// TIA Portal project "MABFactoryIO_Project" (V18)
// TIA Portal - Factory IO

(* hardware
DEVICE "S71500/ET200MP-Station_1"  S7-1500 station
   slot 0: "Profilschiene_0"  Rack  6ES7 590-1***0-0AA0
   slot 1: "PLC_1"  CPU 1517-3 PN/DP  6ES7 517-3AP00-0AB0  V2.6
      slot 3: "CPU-Display_1"  6ES7591-1BA00-0AA0
      slot 32768: "PROFINET-Schnittstelle_1"  X1
         slot 32769: "Port_1"  X1 P1
         slot 32770: "Port_2"  X1 P2
      slot 33024: "PROFINET interface_1"  X2
      slot 33280: "DP interface_1"  X3
   slot 2: "AI 8xU/I/RTD/TC ST_1"  AI 8xU/I/RTD/TC ST  6ES7 531-7KF00-0AB0  V2.0
   slot 3: "AI 8xU/I/RTD/TC ST_2"  AI 8xU/I/RTD/TC ST  6ES7 531-7KF00-0AB0  V2.0
   slot 4: "AI 8xU/I/RTD/TC ST_3"  AI 8xU/I/RTD/TC ST  6ES7 531-7KF00-0AB0  V2.0
   slot 5: "AI 8xU/I/RTD/TC ST_4"  AI 8xU/I/RTD/TC ST  6ES7 531-7KF00-0AB0  V2.0
   slot 6: "DI 16x24VDC BA_1"  DI 16x24VDC BA  6ES7 521-1BH10-0AA0  V1.0
*)

// ===== PLC "PLC_1"  CPU 1517-3 PN/DP =====

VAR_GLOBAL   // PLC tag table "Standard-Variablentabelle"
   "BC-L0" AT %Q10.0 : Bool;
   "BC-L1.1" AT %Q10.1 : Bool;
   "BC-L2" AT %Q10.3 : Bool;
   "BC-L3" AT %Q10.4 : Bool;
   "BC-L4" AT %Q10.5 : Bool;
   "BCS-L0" AT %Q10.6 : Bool;
   "BCS-L1" AT %Q10.7 : Bool;
   "BCC-L0" AT %Q11.0 : Bool;
   "BC-R0" AT %Q11.1 : Bool;
   "BC-R1.1" AT %Q11.2 : Bool;
   "BC-R2" AT %Q11.4 : Bool;
   "BC-R3" AT %Q11.5 : Bool;
   "BCS-R0" AT %Q11.6 : Bool;
   "BCS-R1" AT %Q11.7 : Bool;
   "BCC-R0" AT %Q12.0 : Bool;
   "Conveyor_SR" AT %M10.0 : Bool;
   "Start_Button" AT %I0.0 : Bool;
   "Stop_Button" AT %I0.1 : Bool;
   "BluePileUp" AT %I5.0 : Bool;
   "GreenPileUp" AT %I5.1 : Bool;
   "GreenRawSensor" AT %I4.7 : Bool;
   "BluePileReset" AT %I4.6 : Bool;
   "BC-L1.2" AT %Q10.2 : Bool;
   "BC-R1.2" AT %Q11.3 : Bool;
   "PusherLımıt" AT %I5.2 : Bool;
   "GreenSequenceSensor" AT %I5.3 : Bool;
   "BlueLineSR" AT %M10.1 : Bool;
   "BlueSetter" AT %M1.0 : Bool;
   "GreenLineSR" AT %M10.2 : Bool;
   "GreenSetter" AT %M1.1 : Bool;
   "PusherRight" AT %Q5.0 : Bool;
   "GreenSubline" AT %Q5.1 : Bool;
   "RightLaneBlock" AT %M3.0 : Bool;
   "IsBusy" AT %M3.1 : Bool;
   "SortSR" AT %M10.3 : Bool;
   "SortSR_" AT %M10.4 : Bool;
   "BACUncontrolled" AT %Q3.0 : Bool;
   "BACSBL" AT %Q3.2 : Bool;
   "BSBLeft" AT %Q3.5 : Bool;
   "BACLoadBeltLeft" AT %Q3.3 : Bool;
   "BACLoadBeltRight" AT %Q3.4 : Bool;
   "BACSBR" AT %Q3.1 : Bool;
   "BlueSubline" AT %Q5.2 : Bool;
   "MachineCenterSR" AT %M10.5 : Bool;
   "Machine0" AT %Q0.0 : Bool;
   "Machine1" AT %Q0.1 : Bool;
   "Machine2" AT %Q0.2 : Bool;
   "Machine3" AT %Q0.3 : Bool;
   "Machine0ProduceLids" AT %Q0.4 : Bool;
   "Machine1ProduceLids" AT %Q0.5 : Bool;
   "GreenPileReset" AT %I4.5 : Bool;
   "GreenClosePrevent" AT %I4.4 : Bool;
   "BlueClosePrevent" AT %I4.3 : Bool;
   "MCIsBusy_0" AT %I1.0 : Bool;
   "MCIsBusy_1" AT %I1.1 : Bool;
   "MCIsBusy_2" AT %I1.2 : Bool;
   "MCIsBusy_3" AT %I1.3 : Bool;
   "LPLid_SR" AT %M10.6 : Bool;
   "LPBase_SR" AT %M10.7 : Bool;
   "DiffClampLid" AT %I1.4 : Bool;
   "DiffClampBase" AT %I1.5 : Bool;
   "LPBaseClamped" AT %I1.6 : Bool;
   "LPLidClamped" AT %I1.7 : Bool;
   "LPBaseClamp" AT %Q0.6 : Bool;
   "LPLidClamp" AT %Q0.7 : Bool;
   "TwoAxisDETECT" AT %I2.0 : Bool;
   "TwoAxisDOWN" AT %Q1.0 : Bool;
   "TwoAxisGRAB" AT %Q1.1 : Bool;
   "TwoAxisSR" AT %M11.0 : Bool;
   "LeftPositionerInLim" AT %I2.1 : Bool;
   "TwoAxisFRWD" AT %Q1.2 : Bool;
   "TwoAxisX" AT %I2.2 : Bool;
   "TwoAxisZ" AT %I2.3 : Bool;
   "TwoAxisUPDOWN" AT %I11.1 : Bool;
   "XlimReached" AT %M3.2 : Bool;
   "TwoAxisConnection" AT %M11.2 : Bool;
   "ConnectionComplete" AT %M3.3 : Bool;
   "TwoAxGrabbed" AT %M3.4 : Bool;
   "TwoAxisXSR" AT %M11.1 : Bool;
   "CapTwoAxinPos" AT %I2.4 : Bool;
   "LPRaise" AT %Q1.3 : Bool;
   "LastSR" AT %M11.4 : Bool;
   "CapFullPasse" AT %I2.5 : Bool;
   "AssemblerConvSR" AT %M11.5 : Bool;
   "ACUncontrolled" AT %Q2.0 : Bool;
   "ACFeedBelt" AT %Q2.1 : Bool;
   "ACSBL" AT %Q2.2 : Bool;
   "ACSBR" AT %Q2.3 : Bool;
   "SB_SR" AT %M11.6 : Bool;
   "ACLoadBeltLeft" AT %Q2.4 : Bool;
   "ACLoadBeltRight" AT %Q2.5 : Bool;
   "SBLeft" AT %Q2.6 : Bool;
   "SBRight" AT %Q2.7 : Bool;
   "DiffSBLeft" AT %I2.6 : Bool;
   "DiffSBRight" AT %I2.7 : Bool;
   "CapLoadPassed" AT %I3.0 : Bool;
   "ResetDelay" AT %M11.3 : Bool;
   "LaneFilled" AT %M3.5 : Bool;
   "AssemblerLoaded" AT %M3.6 : Bool;
   "CapBasePassed" AT %I3.1 : Bool;
   "BlueLidSR" AT %M12.0 : Bool;
   "BlueBaseSR" AT %M12.1 : Bool;
   "BlueGrabSR" AT %M12.2 : Bool;
   "BTwoAxForw" AT %M12.3 : Bool;
   "BDiffClampLid" AT %I6.0 : Bool;
   "BDiffClampBase" AT %I6.1 : Bool;
   "BRPBaseClamp" AT %I6.3 : Bool;
   "BLPLidClamped" AT %I6.2 : Bool;
   "BTwoAxDETECT" AT %I6.4 : Bool;
   "BTwoAxisX" AT %I6.5 : Bool;
   "BTwoAxisZ" AT %I6.6 : Bool;
   "BCapFullPassed" AT %I6.7 : Bool;
   "BTwoAxGRAB" AT %Q6.0 : Bool;
   "BRPClamp" AT %Q6.2 : Bool;
   "BLPLidClamp" AT %Q6.1 : Bool;
   "BTwoAxDOWN" AT %Q6.3 : Bool;
   "BTwoAxisFRWD" AT %Q6.4 : Bool;
   "BRPRise" AT %Q6.5 : Bool;
   "BSConvSR" AT %M13.0 : Bool;
   "BAConv_Filled" AT %M13.1 : Bool;
   "BAssemblerLoaded" AT %M3.7 : Bool;
   "BCapLidPassed" AT %I7.1 : Bool;
   "BCapBasePassed" AT %I7.0 : Bool;
   "BSBRight" AT %Q3.6 : Bool;
   "BDiffSBLeft" AT %I7.2 : Bool;
   "BDiffSBRight" AT %I7.3 : Bool;
   "R0 Reset" AT %I0.2 : Bool;
   "Tag_1" AT %M12.7 : Bool;
   "PalletizerSR" AT %M12.4 : Bool;
   "PalletizerPushSR" AT %M12.5 : Bool;
   "DiffPalletizerEntry" AT %I8.0 : Bool;
   "CapPalletizerİnLine" AT %I8.1 : Bool;
   "PalletizerPushLimit" AT %I8.2 : Bool;
   "PalletizerBelt+" AT %Q8.0 : Bool;
   "PalletizerPush" AT %Q8.1 : Bool;
   "CapPalletizerPushİnimit" AT %I8.3 : Bool;
   "CapProdSR" AT %M12.6 : Bool;
   "PalletizerClamped" AT %I8.4 : Bool;
   "PalletizerClamp" AT %Q8.2 : Bool;
END_VAR

// folder: Assembling Operations/BlueProductAssemblyLine

DATA_BLOCK "BlueAssemblerConveyor_DB"   // DB15
{ S7_Optimized_Access := 'TRUE' }
VERSION : 0.1
// stored: InstanceOfName BlueAssemblerConveyor
"BlueAssemblerConveyor"
BEGIN
END_DATA_BLOCK

DATA_BLOCK "BlueAssembler_DB"   // DB16
{ S7_Optimized_Access := 'TRUE' }
VERSION : 0.1
// stored: InstanceOfName BlueAssembler
"BlueAssembler"
BEGIN
END_DATA_BLOCK

DATA_BLOCK "BlueAssemblyReset_DB"   // DB17
{ S7_Optimized_Access := 'TRUE' }
VERSION : 0.1
// stored: InstanceOfName BlueAssemblyReset
"BlueAssemblyReset"
BEGIN
END_DATA_BLOCK

// folder: Assembling Operations/GreenProductAssemblyLine

DATA_BLOCK "Assembler_DB"   // DB4
{ S7_Optimized_Access := 'TRUE' }
VERSION : 0.1
// stored: InstanceOfName Assembler
"Assembler"
BEGIN
END_DATA_BLOCK

DATA_BLOCK "AssemblerConveyor_DB"   // DB6
{ S7_Optimized_Access := 'TRUE' }
VERSION : 0.1
// stored: InstanceOfName AssemblerConveyor
"AssemblerConveyor"
BEGIN
END_DATA_BLOCK

DATA_BLOCK "AssemblyReset_DB"   // DB12
{ S7_Optimized_Access := 'TRUE' }
VERSION : 0.1
// stored: InstanceOfName AssemblyReset
"AssemblyReset"
BEGIN
END_DATA_BLOCK

// folder: Sortıng Operations

DATA_BLOCK "Conveyor_SetLR_DB"   // DB1
{ S7_Optimized_Access := 'TRUE' }
VERSION : 0.1
// stored: InstanceOfName Conveyor_SetLR
"Conveyor_SetLR"
BEGIN
END_DATA_BLOCK

DATA_BLOCK "MachineCenters_DB"   // DB2
{ S7_Optimized_Access := 'TRUE' }
VERSION : 0.1
// stored: InstanceOfName MachineCenters
"MachineCenters"
BEGIN
END_DATA_BLOCK

DATA_BLOCK "SortControl_DB"   // DB3
{ S7_Optimized_Access := 'TRUE' }
VERSION : 0.1
// stored: InstanceOfName SortControl
"SortControl"
BEGIN
END_DATA_BLOCK

// folder: System blocks/Program resources

DATA_BLOCK "liddelay"   // DB5
{ S7_Optimized_Access := 'TRUE' }
AUTHOR : Simatic
FAMILY : IEC
NAME : IEC_TMR
VERSION : 1.0
// stored: InstanceOfName IEC_TIMER
"IEC_TIMER"
BEGIN
END_DATA_BLOCK

DATA_BLOCK "IEC_Timer_0_DB"   // DB7
{ S7_Optimized_Access := 'TRUE' }
AUTHOR : Simatic
FAMILY : IEC
NAME : IEC_TMR
VERSION : 1.0
// stored: InstanceOfName IEC_TIMER
"IEC_TIMER"
BEGIN
END_DATA_BLOCK

DATA_BLOCK "ClampDelay"   // DB8
{ S7_Optimized_Access := 'TRUE' }
AUTHOR : Simatic
FAMILY : IEC
NAME : IEC_TMR
VERSION : 1.0
// stored: InstanceOfName IEC_TIMER
"IEC_TIMER"
BEGIN
END_DATA_BLOCK

DATA_BLOCK "IEC_Timer_0_DB_1"   // DB9
{ S7_Optimized_Access := 'TRUE' }
AUTHOR : Simatic
FAMILY : IEC
NAME : IEC_TMR
VERSION : 1.0
// stored: InstanceOfName IEC_TIMER
"IEC_TIMER"
BEGIN
END_DATA_BLOCK

DATA_BLOCK "IEC_Timer_0_DB_2"   // DB10
{ S7_Optimized_Access := 'TRUE' }
AUTHOR : Simatic
FAMILY : IEC
NAME : IEC_TMR
VERSION : 1.0
// stored: InstanceOfName IEC_TIMER
"IEC_TIMER"
BEGIN
END_DATA_BLOCK

DATA_BLOCK "IEC_Timer_0_DB_3"   // DB11
{ S7_Optimized_Access := 'TRUE' }
AUTHOR : Simatic
FAMILY : IEC
NAME : IEC_TMR
VERSION : 1.0
// stored: InstanceOfName IEC_TIMER
"IEC_TIMER"
BEGIN
END_DATA_BLOCK

DATA_BLOCK "IEC_Timer_0_DB_4"   // DB13
{ S7_Optimized_Access := 'TRUE' }
AUTHOR : Simatic
FAMILY : IEC
NAME : IEC_TMR
VERSION : 1.0
// stored: InstanceOfName IEC_TIMER
"IEC_TIMER"
BEGIN
END_DATA_BLOCK

DATA_BLOCK "IEC_Timer_0_DB_5"   // DB14
{ S7_Optimized_Access := 'TRUE' }
AUTHOR : Simatic
FAMILY : IEC
NAME : IEC_TMR
VERSION : 1.0
// stored: InstanceOfName IEC_TIMER
"IEC_TIMER"
BEGIN
END_DATA_BLOCK

DATA_BLOCK "IEC_Timer_0_DB_6"   // DB18
{ S7_Optimized_Access := 'TRUE' }
AUTHOR : Simatic
FAMILY : IEC
NAME : IEC_TMR
VERSION : 1.0
// stored: InstanceOfName IEC_TIMER
"IEC_TIMER"
BEGIN
END_DATA_BLOCK

DATA_BLOCK "IEC_Timer_0_DB_7"   // DB19
{ S7_Optimized_Access := 'TRUE' }
AUTHOR : Simatic
FAMILY : IEC
NAME : IEC_TMR
VERSION : 1.0
// stored: InstanceOfName IEC_TIMER
"IEC_TIMER"
BEGIN
END_DATA_BLOCK

DATA_BLOCK "IEC_Timer_0_DB_8"   // DB20
{ S7_Optimized_Access := 'TRUE' }
AUTHOR : Simatic
FAMILY : IEC
NAME : IEC_TMR
VERSION : 1.0
// stored: InstanceOfName IEC_TIMER
"IEC_TIMER"
BEGIN
END_DATA_BLOCK

DATA_BLOCK "IEC_Timer_0_DB_9"   // DB21
{ S7_Optimized_Access := 'TRUE' }
AUTHOR : Simatic
FAMILY : IEC
NAME : IEC_TMR
VERSION : 1.0
// stored: InstanceOfName IEC_TIMER
"IEC_TIMER"
BEGIN
END_DATA_BLOCK

DATA_BLOCK "IEC_Timer_0_DB_10"   // DB22
{ S7_Optimized_Access := 'TRUE' }
AUTHOR : Simatic
FAMILY : IEC
NAME : IEC_TMR
VERSION : 1.0
// stored: InstanceOfName IEC_TIMER
"IEC_TIMER"
BEGIN
END_DATA_BLOCK

DATA_BLOCK "IEC_Timer_0_DB_11"   // DB23
{ S7_Optimized_Access := 'TRUE' }
AUTHOR : Simatic
FAMILY : IEC
NAME : IEC_TMR
VERSION : 1.0
// stored: InstanceOfName IEC_TIMER
"IEC_TIMER"
BEGIN
END_DATA_BLOCK

DATA_BLOCK "IEC_Timer_0_DB_12"   // DB24
{ S7_Optimized_Access := 'TRUE' }
AUTHOR : Simatic
FAMILY : IEC
NAME : IEC_TMR
VERSION : 1.0
// stored: InstanceOfName IEC_TIMER
"IEC_TIMER"
BEGIN
END_DATA_BLOCK

DATA_BLOCK "IEC_Timer_0_DB_13"   // DB25
{ S7_Optimized_Access := 'TRUE' }
AUTHOR : Simatic
FAMILY : IEC
NAME : IEC_TMR
VERSION : 1.0
// stored: InstanceOfName IEC_TIMER
"IEC_TIMER"
BEGIN
END_DATA_BLOCK

DATA_BLOCK "IEC_Timer_0_DB_14"   // DB26
{ S7_Optimized_Access := 'TRUE' }
AUTHOR : Simatic
FAMILY : IEC
NAME : IEC_TMR
VERSION : 1.0
// stored: InstanceOfName IEC_TIMER
"IEC_TIMER"
BEGIN
END_DATA_BLOCK

DATA_BLOCK "IEC_Timer_0_DB_15"   // DB27
{ S7_Optimized_Access := 'TRUE' }
AUTHOR : Simatic
FAMILY : IEC
NAME : IEC_TMR
VERSION : 1.0
// stored: InstanceOfName IEC_TIMER
"IEC_TIMER"
BEGIN
END_DATA_BLOCK

// folder: (top level)

FUNCTION "MHJ-PLC-Lab-Function-S71500" : Void   // FC9000, SCL
{ S7_Optimized_Access := 'TRUE' }
VERSION : 0.1
   VAR_TEMP
      Value : Byte;
      ForCounter : Int;
   END_VAR
   VAR CONSTANT
      Value_01_DW : DWord := 16#1223_5486;
      Value_02_DW : DWord := 16#A6C9_D1F5;
   END_VAR
BEGIN

   #Value:=PEEK(area := 16#82,
        dbNumber := 0,
        byteOffset := 511);
   #Value := #Value + 1;

   POKE(area := 16#82,
        dbNumber := 0,
        byteOffset := 511,
        value := #Value);

   POKE(area := 16#82,
        dbNumber := 0,
        byteOffset := 1016,
        value := #Value_01_DW);
   POKE(area := 16#82,
        dbNumber := 0,
        byteOffset := 1020,
        value := #Value_02_DW);

   FOR #ForCounter := 0 TO 63 DO
       #Value:=PEEK(area := 16#1,
            dbNumber := 0,
            byteOffset := #ForCounter);
       POKE(area := 16#81,
            dbNumber := 0,
            byteOffset := #ForCounter,
            value := #Value);
   END_FOR;
   #Value := PEEK(area := 16#1,
                  dbNumber := 0,
                  byteOffset := 512);
   POKE(area := 16#82,
        dbNumber := 0,
        byteOffset := 512,
        value := #Value);
END_FUNCTION

ORGANIZATION_BLOCK "Main"   // OB1, LAD, ProgramCycle
TITLE = "Main Program Sweep (Cycle)"
{ S7_Optimized_Access := 'TRUE' }
VERSION : 0.1
   VAR_INPUT
      Initial_Call : Bool;   // Initial call of this OB
      Remanence : Bool;   // =True, if remanent data are available
   END_VAR
BEGIN

REGION Network 1
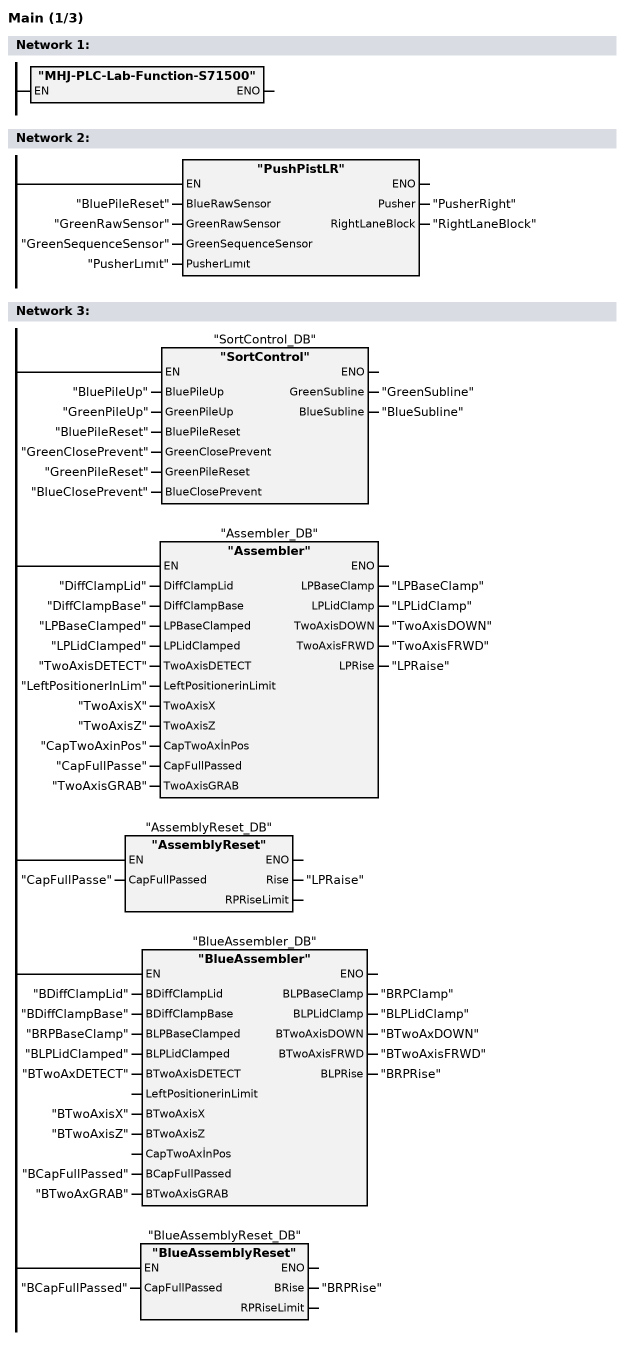
   RUNG wire#powerrail
      "MHJ-PLC-Lab-Function-S71500"()
   END_RUNG
   // the same network as SCL:
   "MHJ-PLC-Lab-Function-S71500"();
END_REGION

REGION Network 2
   RUNG wire#powerrail
      "PushPistLR"(BlueRawSensor := "BluePileReset", GreenRawSensor := "GreenRawSensor", GreenSequenceSensor := "GreenSequenceSensor", PusherLımıt := "PusherLımıt", Pusher => "PusherRight", RightLaneBlock => "RightLaneBlock")
   END_RUNG
   // the same network as SCL:
   "PushPistLR"(BlueRawSensor := "BluePileReset",
                GreenRawSensor := "GreenRawSensor",
                GreenSequenceSensor := "GreenSequenceSensor",
                PusherLımıt := "PusherLımıt",
                Pusher => "PusherRight",
                RightLaneBlock => "RightLaneBlock");
END_REGION

REGION Network 3
   RUNG wire#powerrail
      "SortControl_DB"(BluePileUp := "BluePileUp", GreenPileUp := "GreenPileUp", BluePileReset := "BluePileReset", GreenClosePrevent := "GreenClosePrevent", GreenPileReset := "GreenPileReset", BlueClosePrevent := "BlueClosePrevent", GreenSubline => "GreenSubline", BlueSubline => "BlueSubline")
   END_RUNG
   RUNG wire#powerrail
      "Assembler_DB"(DiffClampLid := "DiffClampLid", DiffClampBase := "DiffClampBase", LPBaseClamped := "LPBaseClamped", LPLidClamped := "LPLidClamped", TwoAxisDETECT := "TwoAxisDETECT", LeftPositionerinLimit := "LeftPositionerInLim", TwoAxisX := "TwoAxisX", TwoAxisZ := "TwoAxisZ", CapTwoAxİnPos := "CapTwoAxinPos", CapFullPassed := "CapFullPasse", TwoAxisGRAB := "TwoAxisGRAB", LPBaseClamp => "LPBaseClamp", LPLidClamp => "LPLidClamp", TwoAxisDOWN => "TwoAxisDOWN", TwoAxisFRWD => "TwoAxisFRWD", LPRise => "LPRaise")
   END_RUNG
   RUNG wire#powerrail
      "AssemblyReset_DB"(CapFullPassed := "CapFullPasse", Rise => "LPRaise", RPRiseLimit =>)
   END_RUNG
   RUNG wire#powerrail
      "BlueAssembler_DB"(BDiffClampLid := "BDiffClampLid", BDiffClampBase := "BDiffClampBase", BLPBaseClamped := "BRPBaseClamp", BLPLidClamped := "BLPLidClamped", BTwoAxisDETECT := "BTwoAxDETECT", LeftPositionerinLimit :=, BTwoAxisX := "BTwoAxisX", BTwoAxisZ := "BTwoAxisZ", CapTwoAxİnPos :=, BCapFullPassed := "BCapFullPassed", BTwoAxisGRAB := "BTwoAxGRAB", BLPBaseClamp => "BRPClamp", BLPLidClamp => "BLPLidClamp", BTwoAxisDOWN => "BTwoAxDOWN", BTwoAxisFRWD => "BTwoAxisFRWD", BLPRise => "BRPRise")
   END_RUNG
   RUNG wire#powerrail
      "BlueAssemblyReset_DB"(CapFullPassed := "BCapFullPassed", BRise => "BRPRise", RPRiseLimit =>)
   END_RUNG
   // the same network as SCL:
   "SortControl_DB"(BluePileUp := "BluePileUp",   // "SortControl"
                    GreenPileUp := "GreenPileUp",
                    BluePileReset := "BluePileReset",
                    GreenClosePrevent := "GreenClosePrevent",
                    GreenPileReset := "GreenPileReset",
                    BlueClosePrevent := "BlueClosePrevent",
                    GreenSubline => "GreenSubline",
                    BlueSubline => "BlueSubline");
   "Assembler_DB"(DiffClampLid := "DiffClampLid",   // "Assembler"
                  DiffClampBase := "DiffClampBase",
                  LPBaseClamped := "LPBaseClamped",
                  LPLidClamped := "LPLidClamped",
                  TwoAxisDETECT := "TwoAxisDETECT",
                  LeftPositionerinLimit := "LeftPositionerInLim",
                  TwoAxisX := "TwoAxisX",
                  TwoAxisZ := "TwoAxisZ",
                  CapTwoAxİnPos := "CapTwoAxinPos",
                  CapFullPassed := "CapFullPasse",
                  TwoAxisGRAB := "TwoAxisGRAB",
                  LPBaseClamp => "LPBaseClamp",
                  LPLidClamp => "LPLidClamp",
                  TwoAxisDOWN => "TwoAxisDOWN",
                  TwoAxisFRWD => "TwoAxisFRWD",
                  LPRise => "LPRaise");
   "AssemblyReset_DB"(CapFullPassed := "CapFullPasse", Rise => "LPRaise");   // "AssemblyReset"
   "BlueAssembler_DB"(BDiffClampLid := "BDiffClampLid",   // "BlueAssembler"
                      BDiffClampBase := "BDiffClampBase",
                      BLPBaseClamped := "BRPBaseClamp",
                      BLPLidClamped := "BLPLidClamped",
                      BTwoAxisDETECT := "BTwoAxDETECT",
                      BTwoAxisX := "BTwoAxisX",
                      BTwoAxisZ := "BTwoAxisZ",
                      BCapFullPassed := "BCapFullPassed",
                      BTwoAxisGRAB := "BTwoAxGRAB",
                      BLPBaseClamp => "BRPClamp",
                      BLPLidClamp => "BLPLidClamp",
                      BTwoAxisDOWN => "BTwoAxDOWN",
                      BTwoAxisFRWD => "BTwoAxisFRWD",
                      BLPRise => "BRPRise");
   "BlueAssemblyReset_DB"(CapFullPassed := "BCapFullPassed", BRise => "BRPRise");   // "BlueAssemblyReset"
END_REGION

REGION Network 4
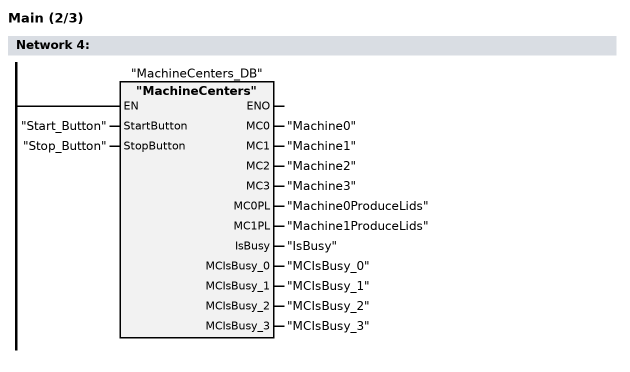
   RUNG wire#powerrail
      "MachineCenters_DB"(StartButton := "Start_Button", StopButton := "Stop_Button", MC0 => "Machine0", MC1 => "Machine1", MC2 => "Machine2", MC3 => "Machine3", MC0PL => "Machine0ProduceLids", MC1PL => "Machine1ProduceLids", IsBusy => "IsBusy", MCIsBusy_0 => "MCIsBusy_0", MCIsBusy_1 => "MCIsBusy_1", MCIsBusy_2 => "MCIsBusy_2", MCIsBusy_3 => "MCIsBusy_3")
   END_RUNG
   // the same network as SCL:
   "MachineCenters_DB"(StartButton := "Start_Button",   // "MachineCenters"
                       StopButton := "Stop_Button",
                       MC0 => "Machine0",
                       MC1 => "Machine1",
                       MC2 => "Machine2",
                       MC3 => "Machine3",
                       MC0PL => "Machine0ProduceLids",
                       MC1PL => "Machine1ProduceLids",
                       IsBusy => "IsBusy",
                       MCIsBusy_0 => "MCIsBusy_0",
                       MCIsBusy_1 => "MCIsBusy_1",
                       MCIsBusy_2 => "MCIsBusy_2",
                       MCIsBusy_3 => "MCIsBusy_3");
END_REGION

REGION Network 5
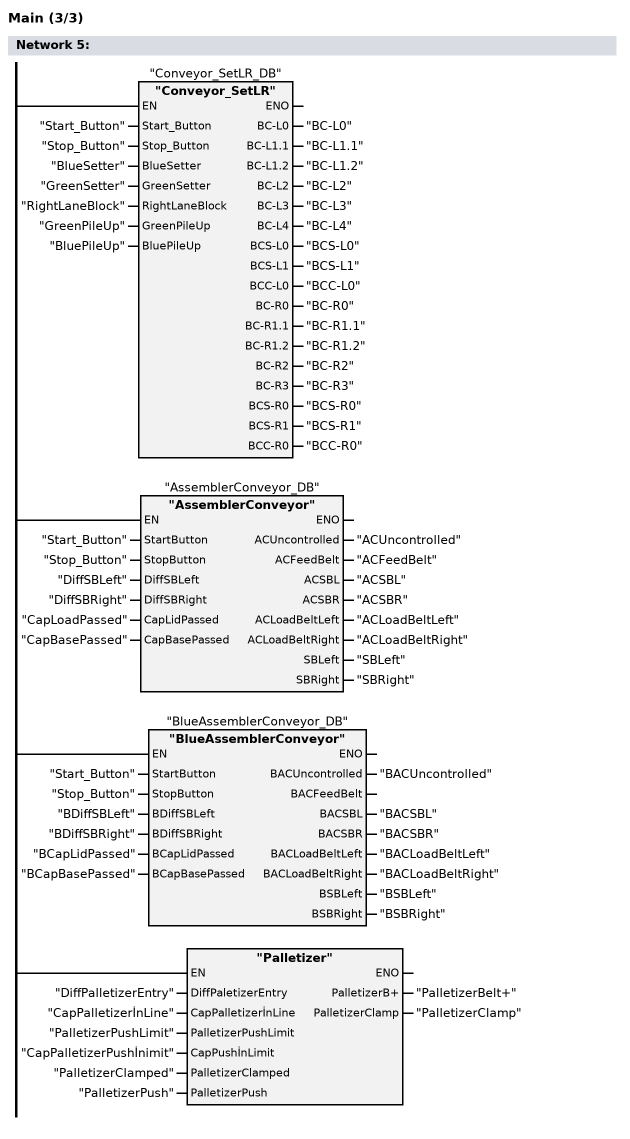
   RUNG wire#powerrail
      "Conveyor_SetLR_DB"(Start_Button := "Start_Button", Stop_Button := "Stop_Button", BlueSetter := "BlueSetter", GreenSetter := "GreenSetter", RightLaneBlock := "RightLaneBlock", GreenPileUp := "GreenPileUp", BluePileUp := "BluePileUp", "BC-L0" => "BC-L0", "BC-L1.1" => "BC-L1.1", "BC-L1.2" => "BC-L1.2", "BC-L2" => "BC-L2", "BC-L3" => "BC-L3", "BC-L4" => "BC-L4", "BCS-L0" => "BCS-L0", "BCS-L1" => "BCS-L1", "BCC-L0" => "BCC-L0", "BC-R0" => "BC-R0", "BC-R1.1" => "BC-R1.1", "BC-R1.2" => "BC-R1.2", "BC-R2" => "BC-R2", "BC-R3" => "BC-R3", "BCS-R0" => "BCS-R0", "BCS-R1" => "BCS-R1", "BCC-R0" => "BCC-R0")
   END_RUNG
   RUNG wire#powerrail
      "AssemblerConveyor_DB"(StartButton := "Start_Button", StopButton := "Stop_Button", DiffSBLeft := "DiffSBLeft", DiffSBRight := "DiffSBRight", CapLidPassed := "CapLoadPassed", CapBasePassed := "CapBasePassed", ACUncontrolled => "ACUncontrolled", ACFeedBelt => "ACFeedBelt", ACSBL => "ACSBL", ACSBR => "ACSBR", ACLoadBeltLeft => "ACLoadBeltLeft", ACLoadBeltRight => "ACLoadBeltRight", SBLeft => "SBLeft", SBRight => "SBRight")
   END_RUNG
   RUNG wire#powerrail
      "BlueAssemblerConveyor_DB"(StartButton := "Start_Button", StopButton := "Stop_Button", BDiffSBLeft := "BDiffSBLeft", BDiffSBRight := "BDiffSBRight", BCapLidPassed := "BCapLidPassed", BCapBasePassed := "BCapBasePassed", BACUncontrolled => "BACUncontrolled", BACFeedBelt =>, BACSBL => "BACSBL", BACSBR => "BACSBR", BACLoadBeltLeft => "BACLoadBeltLeft", BACLoadBeltRight => "BACLoadBeltRight", BSBLeft => "BSBLeft", BSBRight => "BSBRight")
   END_RUNG
   RUNG wire#powerrail
      "Palletizer"(DiffPaletizerEntry := "DiffPalletizerEntry", CapPalletizerİnLine := "CapPalletizerİnLine", PalletizerPushLimit := "PalletizerPushLimit", CapPushİnLimit := "CapPalletizerPushİnimit", PalletizerClamped := "PalletizerClamped", PalletizerPush := "PalletizerPush", "PalletizerB+" => "PalletizerBelt+", PalletizerClamp => "PalletizerClamp")
   END_RUNG
   // the same network as SCL:
   "Conveyor_SetLR_DB"(Start_Button := "Start_Button",   // "Conveyor_SetLR"
                       Stop_Button := "Stop_Button",
                       BlueSetter := "BlueSetter",
                       GreenSetter := "GreenSetter",
                       RightLaneBlock := "RightLaneBlock",
                       GreenPileUp := "GreenPileUp",
                       BluePileUp := "BluePileUp",
                       "BC-L0" => "BC-L0",
                       "BC-L1.1" => "BC-L1.1",
                       "BC-L1.2" => "BC-L1.2",
                       "BC-L2" => "BC-L2",
                       "BC-L3" => "BC-L3",
                       "BC-L4" => "BC-L4",
                       "BCS-L0" => "BCS-L0",
                       "BCS-L1" => "BCS-L1",
                       "BCC-L0" => "BCC-L0",
                       "BC-R0" => "BC-R0",
                       "BC-R1.1" => "BC-R1.1",
                       "BC-R1.2" => "BC-R1.2",
                       "BC-R2" => "BC-R2",
                       "BC-R3" => "BC-R3",
                       "BCS-R0" => "BCS-R0",
                       "BCS-R1" => "BCS-R1",
                       "BCC-R0" => "BCC-R0");
   "AssemblerConveyor_DB"(StartButton := "Start_Button",   // "AssemblerConveyor"
                          StopButton := "Stop_Button",
                          DiffSBLeft := "DiffSBLeft",
                          DiffSBRight := "DiffSBRight",
                          CapLidPassed := "CapLoadPassed",
                          CapBasePassed := "CapBasePassed",
                          ACUncontrolled => "ACUncontrolled",
                          ACFeedBelt => "ACFeedBelt",
                          ACSBL => "ACSBL",
                          ACSBR => "ACSBR",
                          ACLoadBeltLeft => "ACLoadBeltLeft",
                          ACLoadBeltRight => "ACLoadBeltRight",
                          SBLeft => "SBLeft",
                          SBRight => "SBRight");
   "BlueAssemblerConveyor_DB"(StartButton := "Start_Button",   // "BlueAssemblerConveyor"
                           StopButton := "Stop_Button",
                           BDiffSBLeft := "BDiffSBLeft",
                           BDiffSBRight := "BDiffSBRight",
                           BCapLidPassed := "BCapLidPassed",
                           BCapBasePassed := "BCapBasePassed",
                           BACUncontrolled => "BACUncontrolled",
                           BACSBL => "BACSBL",
                           BACSBR => "BACSBR",
                           BACLoadBeltLeft => "BACLoadBeltLeft",
                           BACLoadBeltRight => "BACLoadBeltRight",
                           BSBLeft => "BSBLeft",
                           BSBRight => "BSBRight");
   "Palletizer"(DiffPaletizerEntry := "DiffPalletizerEntry",
                CapPalletizerİnLine := "CapPalletizerİnLine",
                PalletizerPushLimit := "PalletizerPushLimit",
                CapPushİnLimit := "CapPalletizerPushİnimit",
                PalletizerClamped := "PalletizerClamped",
                PalletizerPush := "PalletizerPush",
                "PalletizerB+" => "PalletizerBelt+",
                PalletizerClamp => "PalletizerClamp");
END_REGION
END_ORGANIZATION_BLOCK

// folder: Assembling Operations/BlueProductAssemblyLine

FUNCTION_BLOCK "BlueAssembler"   // FB7, LAD
{ S7_Optimized_Access := 'TRUE' }
VERSION : 0.1
   VAR_INPUT
      BDiffClampLid : Bool;
      BDiffClampBase : Bool;
      BLPBaseClamped : Bool;
      BLPLidClamped : Bool;
      BTwoAxisDETECT : Bool;
      LeftPositionerinLimit : Bool;
      BTwoAxisX : Bool;
      BTwoAxisZ : Bool;
      CapTwoAxİnPos : Bool;
      BCapFullPassed : Bool;
   END_VAR
   VAR_OUTPUT
      BLPBaseClamp : Bool;
      BLPLidClamp : Bool;
      BTwoAxisDOWN : Bool;
      BTwoAxisFRWD : Bool;
      BLPRise : Bool;
   END_VAR
   VAR_IN_OUT
      BTwoAxisGRAB : Bool;
   END_VAR
BEGIN

REGION Network 1
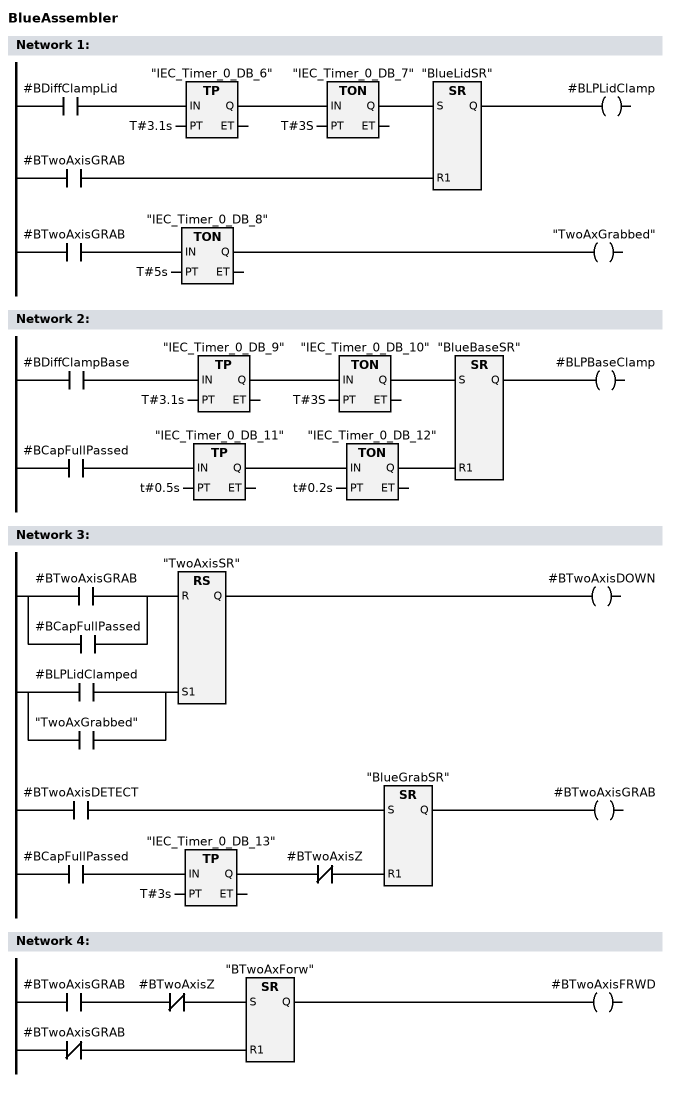
   "IEC_Timer_0_DB_6".TP(IN := #BDiffClampLid, PT := T#3.1s);
   "IEC_Timer_0_DB_7".TON(IN := "IEC_Timer_0_DB_6".Q, PT := T#3S);
   IF "IEC_Timer_0_DB_7".Q THEN
       "BlueLidSR" := TRUE;   // SR flip-flop
   END_IF;
   IF #BTwoAxisGRAB THEN "BlueLidSR" := FALSE; END_IF;
   #BLPLidClamp := "BlueLidSR";
   "IEC_Timer_0_DB_8".TON(IN := #BTwoAxisGRAB, PT := T#5s);
   "TwoAxGrabbed" := "IEC_Timer_0_DB_8".Q;
END_REGION

REGION Network 2
   "IEC_Timer_0_DB_9".TP(IN := #BDiffClampBase, PT := T#3.1s);
   "IEC_Timer_0_DB_10".TON(IN := "IEC_Timer_0_DB_9".Q, PT := T#3S);
   "IEC_Timer_0_DB_11".TP(IN := #BCapFullPassed, PT := t#0.5s);
   "IEC_Timer_0_DB_12".TON(IN := "IEC_Timer_0_DB_11".Q, PT := t#0.2s);
   IF "IEC_Timer_0_DB_10".Q THEN
       "BlueBaseSR" := TRUE;   // SR flip-flop
   END_IF;
   IF "IEC_Timer_0_DB_12".Q THEN "BlueBaseSR" := FALSE; END_IF;
   #BLPBaseClamp := "BlueBaseSR";
END_REGION

REGION Network 3
   IF #BTwoAxisGRAB OR #BCapFullPassed THEN
       "TwoAxisSR" := FALSE;   // RS flip-flop
   END_IF;
   IF #BLPLidClamped OR "TwoAxGrabbed" THEN "TwoAxisSR" := TRUE; END_IF;
   #BTwoAxisDOWN := "TwoAxisSR";
   "IEC_Timer_0_DB_13".TP(IN := #BCapFullPassed, PT := T#3s);
   IF #BTwoAxisDETECT THEN
       "BlueGrabSR" := TRUE;   // SR flip-flop
   END_IF;
   IF "IEC_Timer_0_DB_13".Q AND NOT #BTwoAxisZ THEN "BlueGrabSR" := FALSE; END_IF;
   #BTwoAxisGRAB := "BlueGrabSR";
END_REGION

REGION Network 4
   RUNG wire#powerrail
      Contact( #BTwoAxisGRAB )
      I_Contact( #BTwoAxisZ )
      S_SR(operand := "BTwoAxForw", r1 := wire#w1)
      Coil( #BTwoAxisFRWD )
   END_RUNG
   RUNG wire#powerrail
      I_Contact( #BTwoAxisGRAB )
   END_RUNG wire#w1
   // the same network as SCL:
   IF #BTwoAxisGRAB AND NOT #BTwoAxisZ THEN
       "BTwoAxForw" := TRUE;   // SR flip-flop
   END_IF;
   IF NOT #BTwoAxisGRAB THEN "BTwoAxForw" := FALSE; END_IF;
   #BTwoAxisFRWD := "BTwoAxForw";
END_REGION
END_FUNCTION_BLOCK

FUNCTION_BLOCK "BlueAssemblerConveyor"   // FB8, LAD
{ S7_Optimized_Access := 'TRUE' }
VERSION : 0.1
   VAR_INPUT
      StartButton : Bool;
      StopButton : Bool;
      BDiffSBLeft : Bool;
      BDiffSBRight : Bool;
      BCapLidPassed : Bool;
      BCapBasePassed : Bool;
   END_VAR
   VAR_OUTPUT
      BACUncontrolled : Bool;
      BACFeedBelt : Bool;
      BACSBL : Bool;
      BACSBR : Bool;
      BACLoadBeltLeft : Bool;
      BACLoadBeltRight : Bool;
      BSBLeft : Bool;
      BSBRight : Bool;
   END_VAR
BEGIN

REGION Network 1
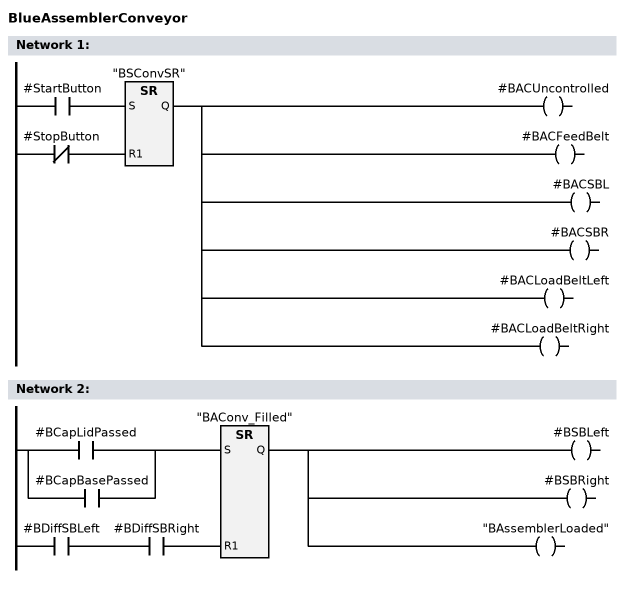
   RUNG wire#powerrail
      Contact( #StartButton )
      S_SR(operand := "BSConvSR", r1 := wire#w1)
      wire#w2
      Coil( #BACUncontrolled )
   END_RUNG
   RUNG wire#powerrail
      I_Contact( #StopButton )
   END_RUNG wire#w1
   RUNG wire#w2
      Coil( #BACFeedBelt )
   END_RUNG
   RUNG wire#w2
      Coil( #BACSBL )
   END_RUNG
   RUNG wire#w2
      Coil( #BACSBR )
   END_RUNG
   RUNG wire#w2
      Coil( #BACLoadBeltLeft )
   END_RUNG
   RUNG wire#w2
      Coil( #BACLoadBeltRight )
   END_RUNG
   // the same network as SCL:
   IF #StartButton THEN
       "BSConvSR" := TRUE;   // SR flip-flop
   END_IF;
   IF NOT #StopButton THEN "BSConvSR" := FALSE; END_IF;
   #BACUncontrolled := "BSConvSR";
   #BACFeedBelt := "BSConvSR";
   #BACSBL := "BSConvSR";
   #BACSBR := "BSConvSR";
   #BACLoadBeltLeft := "BSConvSR";
   #BACLoadBeltRight := "BSConvSR";
END_REGION

REGION Network 2
   RUNG wire#powerrail
      Contact( #BCapLidPassed )
      wire#w1
      S_SR(operand := "BAConv_Filled", r1 := wire#w2)
      wire#w3
      Coil( #BSBLeft )
   END_RUNG
   RUNG wire#powerrail
      Contact( #BCapBasePassed )
   END_RUNG wire#w1
   RUNG wire#powerrail
      Contact( #BDiffSBLeft )
      Contact( #BDiffSBRight )
   END_RUNG wire#w2
   RUNG wire#w3
      Coil( #BSBRight )
   END_RUNG
   RUNG wire#w3
      Coil( "BAssemblerLoaded" )
   END_RUNG
   // the same network as SCL:
   IF #BCapLidPassed OR #BCapBasePassed THEN
       "BAConv_Filled" := TRUE;   // SR flip-flop
   END_IF;
   IF #BDiffSBLeft AND #BDiffSBRight THEN "BAConv_Filled" := FALSE; END_IF;
   #BSBLeft := "BAConv_Filled";
   #BSBRight := "BAConv_Filled";
   "BAssemblerLoaded" := "BAConv_Filled";
END_REGION
END_FUNCTION_BLOCK

FUNCTION_BLOCK "BlueAssemblyReset"   // FB9, LAD
{ S7_Optimized_Access := 'TRUE' }
VERSION : 0.1
   VAR_INPUT
      CapFullPassed : Bool;
   END_VAR
   VAR_OUTPUT
      BRise : Bool;
      RPRiseLimit : Bool;
   END_VAR
BEGIN

REGION Network 1
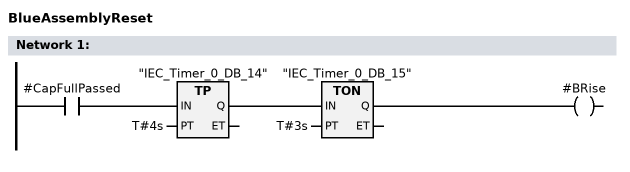
   "IEC_Timer_0_DB_14".TP(IN := #CapFullPassed, PT := T#4s);
   "IEC_Timer_0_DB_15".TON(IN := "IEC_Timer_0_DB_14".Q, PT := T#3s);
   #BRise := "IEC_Timer_0_DB_15".Q;
END_REGION
END_FUNCTION_BLOCK

// folder: Assembling Operations/GreenProductAssemblyLine

FUNCTION_BLOCK "Assembler"   // FB4, LAD
{ S7_Optimized_Access := 'TRUE' }
VERSION : 0.1
   VAR_INPUT
      DiffClampLid : Bool;
      DiffClampBase : Bool;
      LPBaseClamped : Bool;
      LPLidClamped : Bool;
      TwoAxisDETECT : Bool;
      LeftPositionerinLimit : Bool;
      TwoAxisX : Bool;
      TwoAxisZ : Bool;
      CapTwoAxİnPos : Bool;
      CapFullPassed : Bool;
   END_VAR
   VAR_OUTPUT
      LPBaseClamp : Bool;
      LPLidClamp : Bool;
      TwoAxisDOWN : Bool;
      TwoAxisFRWD : Bool;
      LPRise : Bool;
   END_VAR
   VAR_IN_OUT
      TwoAxisGRAB : Bool;
   END_VAR
BEGIN

REGION Network 1
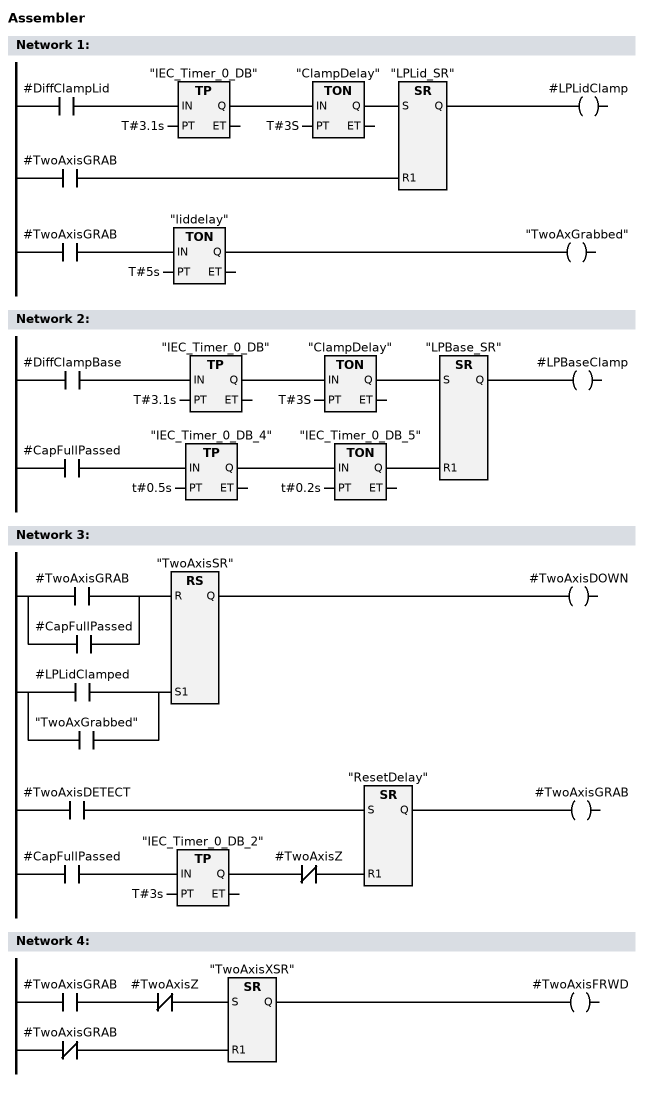
   "IEC_Timer_0_DB".TP(IN := #DiffClampLid, PT := T#3.1s);
   "ClampDelay".TON(IN := "IEC_Timer_0_DB".Q, PT := T#3S);
   IF "ClampDelay".Q THEN
       "LPLid_SR" := TRUE;   // SR flip-flop
   END_IF;
   IF #TwoAxisGRAB THEN "LPLid_SR" := FALSE; END_IF;
   #LPLidClamp := "LPLid_SR";
   "liddelay".TON(IN := #TwoAxisGRAB, PT := T#5s);
   "TwoAxGrabbed" := "liddelay".Q;
END_REGION

REGION Network 2
   "IEC_Timer_0_DB".TP(IN := #DiffClampBase, PT := T#3.1s);
   "ClampDelay".TON(IN := "IEC_Timer_0_DB".Q, PT := T#3S);
   "IEC_Timer_0_DB_4".TP(IN := #CapFullPassed, PT := t#0.5s);
   "IEC_Timer_0_DB_5".TON(IN := "IEC_Timer_0_DB_4".Q, PT := t#0.2s);
   IF "ClampDelay".Q THEN
       "LPBase_SR" := TRUE;   // SR flip-flop
   END_IF;
   IF "IEC_Timer_0_DB_5".Q THEN "LPBase_SR" := FALSE; END_IF;
   #LPBaseClamp := "LPBase_SR";
END_REGION

REGION Network 3
   IF #TwoAxisGRAB OR #CapFullPassed THEN
       "TwoAxisSR" := FALSE;   // RS flip-flop
   END_IF;
   IF #LPLidClamped OR "TwoAxGrabbed" THEN "TwoAxisSR" := TRUE; END_IF;
   #TwoAxisDOWN := "TwoAxisSR";
   "IEC_Timer_0_DB_2".TP(IN := #CapFullPassed, PT := T#3s);
   IF #TwoAxisDETECT THEN
       "ResetDelay" := TRUE;   // SR flip-flop
   END_IF;
   IF "IEC_Timer_0_DB_2".Q AND NOT #TwoAxisZ THEN "ResetDelay" := FALSE; END_IF;
   #TwoAxisGRAB := "ResetDelay";
END_REGION

REGION Network 4
   RUNG wire#powerrail
      Contact( #TwoAxisGRAB )
      I_Contact( #TwoAxisZ )
      S_SR(operand := "TwoAxisXSR", r1 := wire#w1)
      Coil( #TwoAxisFRWD )
   END_RUNG
   RUNG wire#powerrail
      I_Contact( #TwoAxisGRAB )
   END_RUNG wire#w1
   // the same network as SCL:
   IF #TwoAxisGRAB AND NOT #TwoAxisZ THEN
       "TwoAxisXSR" := TRUE;   // SR flip-flop
   END_IF;
   IF NOT #TwoAxisGRAB THEN "TwoAxisXSR" := FALSE; END_IF;
   #TwoAxisFRWD := "TwoAxisXSR";
END_REGION
END_FUNCTION_BLOCK

FUNCTION_BLOCK "AssemblerConveyor"   // FB5, LAD
{ S7_Optimized_Access := 'TRUE' }
VERSION : 0.1
   VAR_INPUT
      StartButton : Bool;
      StopButton : Bool;
      DiffSBLeft : Bool;
      DiffSBRight : Bool;
      CapLidPassed : Bool;
      CapBasePassed : Bool;
   END_VAR
   VAR_OUTPUT
      ACUncontrolled : Bool;
      ACFeedBelt : Bool;
      ACSBL : Bool;
      ACSBR : Bool;
      ACLoadBeltLeft : Bool;
      ACLoadBeltRight : Bool;
      SBLeft : Bool;
      SBRight : Bool;
   END_VAR
BEGIN

REGION Network 1
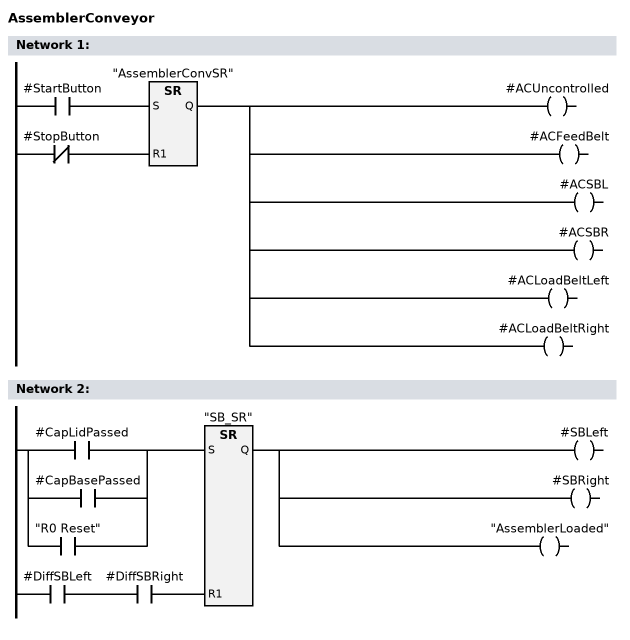
   RUNG wire#powerrail
      Contact( #StartButton )
      S_SR(operand := "AssemblerConvSR", r1 := wire#w1)
      wire#w2
      Coil( #ACUncontrolled )
   END_RUNG
   RUNG wire#powerrail
      I_Contact( #StopButton )
   END_RUNG wire#w1
   RUNG wire#w2
      Coil( #ACFeedBelt )
   END_RUNG
   RUNG wire#w2
      Coil( #ACSBL )
   END_RUNG
   RUNG wire#w2
      Coil( #ACSBR )
   END_RUNG
   RUNG wire#w2
      Coil( #ACLoadBeltLeft )
   END_RUNG
   RUNG wire#w2
      Coil( #ACLoadBeltRight )
   END_RUNG
   // the same network as SCL:
   IF #StartButton THEN
       "AssemblerConvSR" := TRUE;   // SR flip-flop
   END_IF;
   IF NOT #StopButton THEN "AssemblerConvSR" := FALSE; END_IF;
   #ACUncontrolled := "AssemblerConvSR";
   #ACFeedBelt := "AssemblerConvSR";
   #ACSBL := "AssemblerConvSR";
   #ACSBR := "AssemblerConvSR";
   #ACLoadBeltLeft := "AssemblerConvSR";
   #ACLoadBeltRight := "AssemblerConvSR";
END_REGION

REGION Network 2
   RUNG wire#powerrail
      Contact( #CapLidPassed )
      wire#w1
      S_SR(operand := "SB_SR", r1 := wire#w2)
      wire#w3
      Coil( #SBLeft )
   END_RUNG
   RUNG wire#powerrail
      Contact( #CapBasePassed )
   END_RUNG wire#w1
   RUNG wire#powerrail
      Contact( "R0 Reset" )
   END_RUNG wire#w1
   RUNG wire#powerrail
      Contact( #DiffSBLeft )
      Contact( #DiffSBRight )
   END_RUNG wire#w2
   RUNG wire#w3
      Coil( #SBRight )
   END_RUNG
   RUNG wire#w3
      Coil( "AssemblerLoaded" )
   END_RUNG
   // the same network as SCL:
   IF #CapLidPassed OR #CapBasePassed OR "R0 Reset" THEN
       "SB_SR" := TRUE;   // SR flip-flop
   END_IF;
   IF #DiffSBLeft AND #DiffSBRight THEN "SB_SR" := FALSE; END_IF;
   #SBLeft := "SB_SR";
   #SBRight := "SB_SR";
   "AssemblerLoaded" := "SB_SR";
END_REGION
END_FUNCTION_BLOCK

FUNCTION_BLOCK "AssemblyReset"   // FB6, LAD
{ S7_Optimized_Access := 'TRUE' }
VERSION : 0.1
   VAR_INPUT
      CapFullPassed : Bool;
   END_VAR
   VAR_OUTPUT
      Rise : Bool;
      RPRiseLimit : Bool;
   END_VAR
BEGIN

REGION Network 1
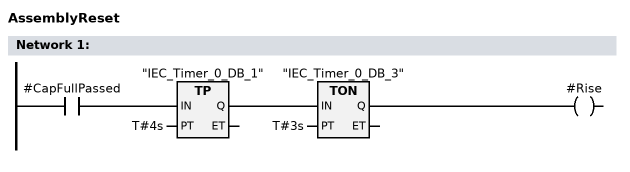
   "IEC_Timer_0_DB_1".TP(IN := #CapFullPassed, PT := T#4s);
   "IEC_Timer_0_DB_3".TON(IN := "IEC_Timer_0_DB_1".Q, PT := T#3s);
   #Rise := "IEC_Timer_0_DB_3".Q;
END_REGION
END_FUNCTION_BLOCK

// folder: Palletizer Operations

FUNCTION "Palletizer" : Void   // FC1, LAD
{ S7_Optimized_Access := 'TRUE' }
VERSION : 0.1
   VAR_INPUT
      DiffPaletizerEntry : Bool;
      CapPalletizerİnLine : Bool;
      PalletizerPushLimit : Bool;
      CapPushİnLimit : Bool;
      PalletizerClamped : Bool;
   END_VAR
   VAR_OUTPUT
      "PalletizerB+" : Bool;
      PalletizerClamp : Bool;
   END_VAR
   VAR_IN_OUT
      PalletizerPush : Bool;
   END_VAR
BEGIN

REGION Network 1
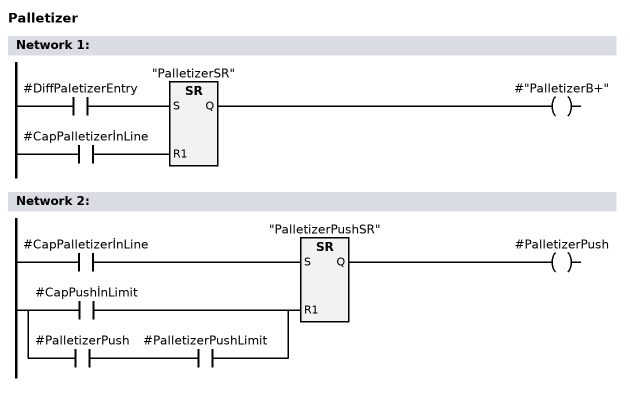
   RUNG wire#powerrail
      Contact( #DiffPaletizerEntry )
      S_SR(operand := "PalletizerSR", r1 := wire#w1)
      Coil( #"PalletizerB+" )
   END_RUNG
   RUNG wire#powerrail
      Contact( #CapPalletizerİnLine )
   END_RUNG wire#w1
   // the same network as SCL:
   IF #DiffPaletizerEntry THEN
       "PalletizerSR" := TRUE;   // SR flip-flop
   END_IF;
   IF #CapPalletizerİnLine THEN "PalletizerSR" := FALSE; END_IF;
   #"PalletizerB+" := "PalletizerSR";
END_REGION

REGION Network 2
   RUNG wire#powerrail
      Contact( #CapPalletizerİnLine )
      S_SR(operand := "PalletizerPushSR", r1 := wire#w1)
      Coil( #PalletizerPush )
   END_RUNG
   RUNG wire#powerrail
      Contact( #CapPushİnLimit )
   END_RUNG wire#w1
   RUNG wire#powerrail
      Contact( #PalletizerPush )
      Contact( #PalletizerPushLimit )
   END_RUNG wire#w1
   // the same network as SCL:
   IF #CapPalletizerİnLine THEN
       "PalletizerPushSR" := TRUE;   // SR flip-flop
   END_IF;
   IF #CapPushİnLimit OR (#PalletizerPush AND #PalletizerPushLimit) THEN "PalletizerPushSR" := FALSE; END_IF;
   #PalletizerPush := "PalletizerPushSR";
END_REGION
END_FUNCTION

// folder: Sortıng Operations

FUNCTION_BLOCK "Conveyor_SetLR"   // FB1, LAD
{ S7_Optimized_Access := 'TRUE' }
VERSION : 0.1
   VAR_INPUT
      Start_Button : Bool;
      Stop_Button : Bool;
      BlueSetter : Bool;
      GreenSetter : Bool;
      RightLaneBlock : Bool;
      GreenPileUp : Bool;
      BluePileUp : Bool;
   END_VAR
   VAR_OUTPUT
      "BC-L0" : Bool;
      "BC-L1.1" : Bool;
      "BC-L1.2" : Bool;
      "BC-L2" : Bool;
      "BC-L3" : Bool;
      "BC-L4" : Bool;
      "BCS-L0" : Bool;
      "BCS-L1" : Bool;
      "BCC-L0" : Bool;
      "BC-R0" : Bool;
      "BC-R1.1" : Bool;
      "BC-R1.2" : Bool;
      "BC-R2" : Bool;
      "BC-R3" : Bool;
      "BCS-R0" : Bool;
      "BCS-R1" : Bool;
      "BCC-R0" : Bool;
   END_VAR
BEGIN

REGION Network 1: LeftConv_CTRL
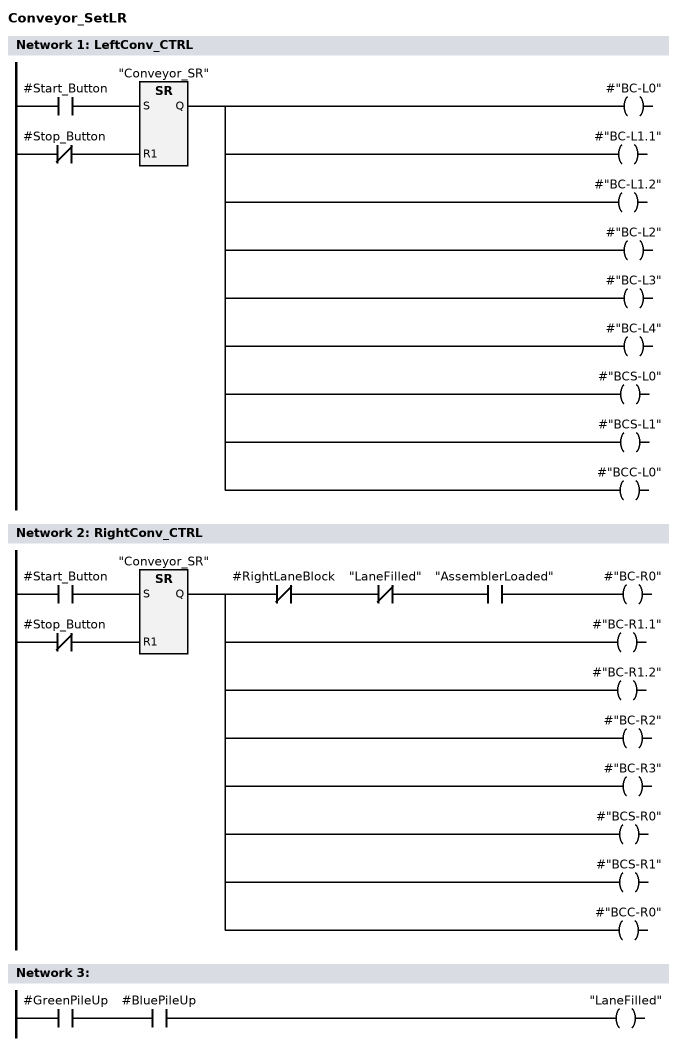
   RUNG wire#powerrail
      Contact( #Start_Button )
      S_SR(operand := "Conveyor_SR", r1 := wire#w1)
      wire#w2
      Coil( #"BC-L0" )
   END_RUNG
   RUNG wire#powerrail
      I_Contact( #Stop_Button )
   END_RUNG wire#w1
   RUNG wire#w2
      Coil( #"BC-L1.1" )
   END_RUNG
   RUNG wire#w2
      Coil( #"BC-L1.2" )
   END_RUNG
   RUNG wire#w2
      Coil( #"BC-L2" )
   END_RUNG
   RUNG wire#w2
      Coil( #"BC-L3" )
   END_RUNG
   RUNG wire#w2
      Coil( #"BC-L4" )
   END_RUNG
   RUNG wire#w2
      Coil( #"BCS-L0" )
   END_RUNG
   RUNG wire#w2
      Coil( #"BCS-L1" )
   END_RUNG
   RUNG wire#w2
      Coil( #"BCC-L0" )
   END_RUNG
   // the same network as SCL:
   IF #Start_Button THEN
       "Conveyor_SR" := TRUE;   // SR flip-flop
   END_IF;
   IF NOT #Stop_Button THEN "Conveyor_SR" := FALSE; END_IF;
   #"BC-L0" := "Conveyor_SR";
   #"BC-L1.1" := "Conveyor_SR";
   #"BC-L1.2" := "Conveyor_SR";
   #"BC-L2" := "Conveyor_SR";
   #"BC-L3" := "Conveyor_SR";
   #"BC-L4" := "Conveyor_SR";
   #"BCS-L0" := "Conveyor_SR";
   #"BCS-L1" := "Conveyor_SR";
   #"BCC-L0" := "Conveyor_SR";
END_REGION

REGION Network 2: RightConv_CTRL
   RUNG wire#powerrail
      Contact( #Start_Button )
      S_SR(operand := "Conveyor_SR", r1 := wire#w1)
      wire#w2
      I_Contact( #RightLaneBlock )
      I_Contact( "LaneFilled" )
      Contact( "AssemblerLoaded" )
      Coil( #"BC-R0" )
   END_RUNG
   RUNG wire#powerrail
      I_Contact( #Stop_Button )
   END_RUNG wire#w1
   RUNG wire#w2
      Coil( #"BC-R1.1" )
   END_RUNG
   RUNG wire#w2
      Coil( #"BC-R1.2" )
   END_RUNG
   RUNG wire#w2
      Coil( #"BC-R2" )
   END_RUNG
   RUNG wire#w2
      Coil( #"BC-R3" )
   END_RUNG
   RUNG wire#w2
      Coil( #"BCS-R0" )
   END_RUNG
   RUNG wire#w2
      Coil( #"BCS-R1" )
   END_RUNG
   RUNG wire#w2
      Coil( #"BCC-R0" )
   END_RUNG
   // the same network as SCL:
   IF #Start_Button THEN
       "Conveyor_SR" := TRUE;   // SR flip-flop
   END_IF;
   IF NOT #Stop_Button THEN "Conveyor_SR" := FALSE; END_IF;
   #"BC-R0" := "Conveyor_SR" AND NOT #RightLaneBlock AND NOT "LaneFilled" AND "AssemblerLoaded";
   #"BC-R1.1" := "Conveyor_SR";
   #"BC-R1.2" := "Conveyor_SR";
   #"BC-R2" := "Conveyor_SR";
   #"BC-R3" := "Conveyor_SR";
   #"BCS-R0" := "Conveyor_SR";
   #"BCS-R1" := "Conveyor_SR";
   #"BCC-R0" := "Conveyor_SR";
END_REGION

REGION Network 3
   RUNG wire#powerrail
      Contact( #GreenPileUp )
      Contact( #BluePileUp )
      Coil( "LaneFilled" )
   END_RUNG
   // the same network as SCL:
   "LaneFilled" := #GreenPileUp AND #BluePileUp;
END_REGION
END_FUNCTION_BLOCK

FUNCTION_BLOCK "SortControl"   // FB2, LAD
{ S7_Optimized_Access := 'TRUE' }
VERSION : 0.1
   VAR_INPUT
      BluePileUp : Bool;
      GreenPileUp : Bool;
      BluePileReset : Bool;
      GreenClosePrevent : Bool;
      GreenPileReset : Bool;
      BlueClosePrevent : Bool;
   END_VAR
   VAR_OUTPUT
      GreenSubline : Bool;
      BlueSubline : Bool;
   END_VAR
BEGIN

REGION Network 1
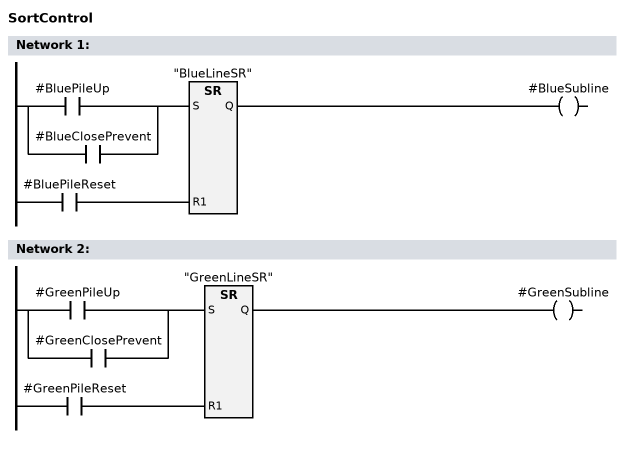
   RUNG wire#powerrail
      Contact( #BluePileUp )
      wire#w1
      S_SR(operand := "BlueLineSR", r1 := wire#w2)
      Coil( #BlueSubline )
   END_RUNG
   RUNG wire#powerrail
      Contact( #BlueClosePrevent )
   END_RUNG wire#w1
   RUNG wire#powerrail
      Contact( #BluePileReset )
   END_RUNG wire#w2
   // the same network as SCL:
   IF #BluePileUp OR #BlueClosePrevent THEN
       "BlueLineSR" := TRUE;   // SR flip-flop
   END_IF;
   IF #BluePileReset THEN "BlueLineSR" := FALSE; END_IF;
   #BlueSubline := "BlueLineSR";
END_REGION

REGION Network 2
   RUNG wire#powerrail
      Contact( #GreenPileUp )
      wire#w1
      S_SR(operand := "GreenLineSR", r1 := wire#w2)
      Coil( #GreenSubline )
   END_RUNG
   RUNG wire#powerrail
      Contact( #GreenClosePrevent )
   END_RUNG wire#w1
   RUNG wire#powerrail
      Contact( #GreenPileReset )
   END_RUNG wire#w2
   // the same network as SCL:
   IF #GreenPileUp OR #GreenClosePrevent THEN
       "GreenLineSR" := TRUE;   // SR flip-flop
   END_IF;
   IF #GreenPileReset THEN "GreenLineSR" := FALSE; END_IF;
   #GreenSubline := "GreenLineSR";
END_REGION
END_FUNCTION_BLOCK

FUNCTION_BLOCK "MachineCenters"   // FB3, LAD
{ S7_Optimized_Access := 'TRUE' }
VERSION : 0.1
   VAR_INPUT
      StartButton : Bool;
      StopButton : Bool;
   END_VAR
   VAR_OUTPUT
      MC0 : Bool;
      MC1 : Bool;
      MC2 : Bool;
      MC3 : Bool;
      MC0PL : Bool;
      MC1PL : Bool;
      IsBusy : Bool;
      MCIsBusy_0 : Bool;
      MCIsBusy_1 : Bool;
      MCIsBusy_2 : Bool;
      MCIsBusy_3 : Bool;
   END_VAR
BEGIN

REGION Network 1
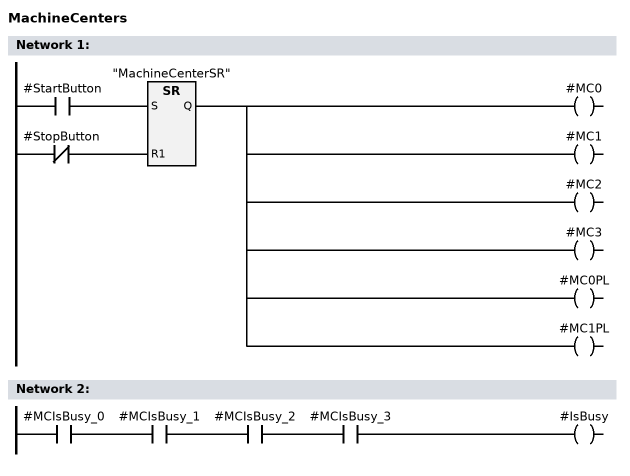
   RUNG wire#powerrail
      Contact( #StartButton )
      S_SR(operand := "MachineCenterSR", r1 := wire#w1)
      wire#w2
      Coil( #MC0 )
   END_RUNG
   RUNG wire#powerrail
      I_Contact( #StopButton )
   END_RUNG wire#w1
   RUNG wire#w2
      Coil( #MC1 )
   END_RUNG
   RUNG wire#w2
      Coil( #MC2 )
   END_RUNG
   RUNG wire#w2
      Coil( #MC3 )
   END_RUNG
   RUNG wire#w2
      Coil( #MC0PL )
   END_RUNG
   RUNG wire#w2
      Coil( #MC1PL )
   END_RUNG
   // the same network as SCL:
   IF #StartButton THEN
       "MachineCenterSR" := TRUE;   // SR flip-flop
   END_IF;
   IF NOT #StopButton THEN "MachineCenterSR" := FALSE; END_IF;
   #MC0 := "MachineCenterSR";
   #MC1 := "MachineCenterSR";
   #MC2 := "MachineCenterSR";
   #MC3 := "MachineCenterSR";
   #MC0PL := "MachineCenterSR";
   #MC1PL := "MachineCenterSR";
END_REGION

REGION Network 2
   RUNG wire#powerrail
      Contact( #MCIsBusy_0 )
      Contact( #MCIsBusy_1 )
      Contact( #MCIsBusy_2 )
      Contact( #MCIsBusy_3 )
      Coil( #IsBusy )
   END_RUNG
   // the same network as SCL:
   #IsBusy := #MCIsBusy_0 AND #MCIsBusy_1 AND #MCIsBusy_2 AND #MCIsBusy_3;
END_REGION
END_FUNCTION_BLOCK

FUNCTION "PushPistLR" : Void   // FC2, LAD
{ S7_Optimized_Access := 'TRUE' }
VERSION : 0.1
   VAR_INPUT
      BlueRawSensor : Bool;
      GreenRawSensor : Bool;
      GreenSequenceSensor : Bool;
      PusherLımıt : Bool;
   END_VAR
   VAR_OUTPUT
      Pusher : Bool;
      RightLaneBlock : Bool;
   END_VAR
BEGIN

REGION Network 1
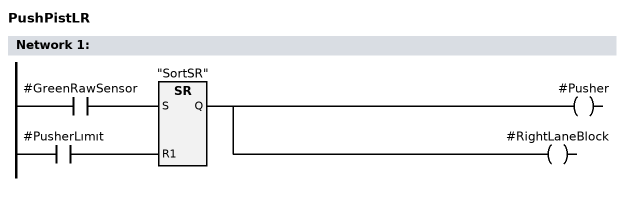
   RUNG wire#powerrail
      Contact( #GreenRawSensor )
      S_SR(operand := "SortSR", r1 := wire#w1)
      wire#w2
      Coil( #Pusher )
   END_RUNG
   RUNG wire#powerrail
      Contact( #PusherLımıt )
   END_RUNG wire#w1
   RUNG wire#w2
      Coil( #RightLaneBlock )
   END_RUNG
   // the same network as SCL:
   IF #GreenRawSensor THEN
       "SortSR" := TRUE;   // SR flip-flop
   END_IF;
   IF #PusherLımıt THEN "SortSR" := FALSE; END_IF;
   #Pusher := "SortSR";
   #RightLaneBlock := "SortSR";
END_REGION
END_FUNCTION